TYPE SM_HMI_ocmd :
STRUCT
  Abort : BOOL;
  Home : BOOL;
  Start : BOOL;
  Stop : BOOL;
  Pause : BOOL;
  Proceed : BOOL;
  Retry : BOOL;
  ActiveStatePermBypass : BOOL;
END_STRUCT
END_TYPE

(* stored: Version 1.1.0.1, ProductVersion 3.1.4024.13
   DUT SM_HMI_ocmd: Id {4f8f7d01-08be-4553-80ff-bed9cd1cb616} *)
